SUBAPPLICATION Uebung_071 (* WBSD auf UT ausgeben, Q1 Schalten wenn Speed &gt;0 *)
  (* Standard: 61499-2 *)
  (* Version 1.0, 2023-10-23, franz *)
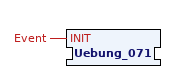
  EVENT_INPUT
    INIT;
  END_EVENT
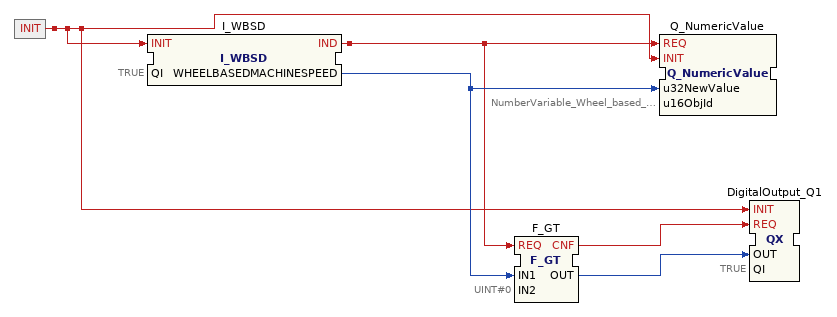
  FBS
    I_WBSD : I_WBSD(QI := TRUE);
    Q_NumericValue : Q_NumericValue(u16ObjId := NumberVariable_Wheel_based_machine_speed);
    DigitalOutput_Q1 : QX(QI := TRUE);
    F_GT : F_GT(IN2 := UINT#0);
  END_FBS
  EVENT_CONNECTIONS
    I_WBSD.IND TO Q_NumericValue.REQ;
    INIT TO I_WBSD.INIT;
    INIT TO Q_NumericValue.INIT;
    INIT TO DigitalOutput_Q1.INIT;
    I_WBSD.IND TO F_GT.REQ;
    F_GT.CNF TO DigitalOutput_Q1.REQ;
  END_CONNECTIONS
  DATA_CONNECTIONS
    I_WBSD.WHEELBASEDMACHINESPEED TO Q_NumericValue.u32NewValue;
    I_WBSD.WHEELBASEDMACHINESPEED TO F_GT.IN1;
    F_GT.OUT TO DigitalOutput_Q1.OUT;
  END_CONNECTIONS
END_SUBAPPLICATION
